LIN {X 0,Y 104.567,Z 489.465,A -85,B 0,C 180,E1 -28252.275,E2 -28252.275} C_VEL
LIN {X 0,Y 104.619,Z 487.581,A -85,B 0,C 180,E1 -28260,E2 -28260} C_VEL
LIN {X 0,Y 104.221,Z 489.218,A -85,B 0,C 180,E1 -28267.958,E2 -28267.958} C_VEL
LIN {X 0,Y 104.511,Z 490.279,A -85,B 0,C 180,E1 -28271.639,E2 -28271.639} C_VEL
LIN {X 0,Y 105.02,Z 492.985,A -85,B 0,C 180,E1 -28277.526,E2 -28277.526} C_VEL
LIN {X 0,Y 105.625,Z 496.885,A -85,B 0,C 180,E1 -28283.53,E2 -28283.53} C_VEL
LIN {X 0,Y 106.054,Z 500.091,A -85,B 0,C 180,E1 -28287.638,E2 -28287.638} C_VEL
LIN {X 0,Y 105.786,Z 504.564,A -85,B 0,C 180,E1 -28292.106,E2 -28292.106} C_VEL
LIN {X 0,Y 104.952,Z 508.015,A -85,B 0,C 180,E1 -28294.982,E2 -28294.982} C_VEL
LIN {X 0,Y 103.687,Z 511.068,A -85,B 0,C 180,E1 -28297.21,E2 -28297.21} C_VEL
LIN {X 0,Y 97.623,Z 518.073,A -85,B 0,C 180,E1 -28300.895,E2 -28300.895} C_VEL
LIN {X 0,Y 90.769,Z 524.928,A -85,B 0,C 180,E1 -28305.826,E2 -28305.826} C_VEL
LIN {X 0,Y 83.786,Z 531.001,A -85,B 0,C 180,E1 -28312.143,E2 -28312.143} C_VEL
LIN {X 0,Y 77.697,Z 535.939,A -85,B 0,C 180,E1 -28320.166,E2 -28320.166} C_VEL
LIN {X 0,Y 73.855,Z 538.844,A -85,B 0,C 180,E1 -28327.627,E2 -28327.627} C_VEL
LIN {X 0,Y 72.25,Z 540.013,A -85,B 0,C 180,E1 -28332.13,E2 -28332.13} C_VEL
LIN {X 0,Y 70.44,Z 541.017,A -85,B 0,C 180,E1 -28336.574,E2 -28336.574} C_VEL
LIN {X 0,Y 68.078,Z 541.734,A -85,B 0,C 180,E1 -28341.053,E2 -28341.053} C_VEL
LIN {X 0,Y 63.796,Z 542.259,A -85,B 0,C 180,E1 -28350.796,E2 -28350.796} C_VEL
LIN {X 0,Y 62.993,Z 542.058,A -85,B 0,C 180,E1 -28356.152,E2 -28356.152} C_VEL
LIN {X 0,Y 63.07,Z 541.9,A -85,B 0,C 180,E1 -28357.958,E2 -28357.958} C_VEL
LIN {X 0,Y 65.242,Z 540.489,A -85,B 0,C 180,E1 -28368.855,E2 -28368.855} C_VEL
LIN {X 0,Y 67.337,Z 539.131,A -85,B 0,C 180,E1 -28374.676,E2 -28374.676} C_VEL
LIN {X 0,Y 71.589,Z 536.26,A -85,B 0,C 180,E1 -28382.681,E2 -28382.681} C_VEL
LIN {X 0,Y 76.937,Z 532.366,A -85,B 0,C 180,E1 -28389.75,E2 -28389.75} C_VEL
LIN {X 0,Y 83.424,Z 527.333,A -85,B 0,C 180,E1 -28395.733,E2 -28395.733} C_VEL
LIN {X 0,Y 90.544,Z 520.995,A -85,B 0,C 180,E1 -28400.915,E2 -28400.915} C_VEL
LIN {X 0,Y 98.183,Z 513.072,A -85,B 0,C 180,E1 -28405.405,E2 -28405.405} C_VEL
LIN {X 0,Y 99.078,Z 511.615,A -85,B 0,C 180,E1 -28406.459,E2 -28406.459} C_VEL
LIN {X 0,Y 100.27,Z 508.389,A -85,B 0,C 180,E1 -28409.327,E2 -28409.327} C_VEL
LIN {X 0,Y 100.77,Z 505.026,A -85,B 0,C 180,E1 -28413.044,E2 -28413.044} C_VEL
LIN {X 0,Y 100.847,Z 503.301,A -85,B 0,C 180,E1 -28415.283,E2 -28415.283} C_VEL
LIN {X 0,Y 100.697,Z 500.442,A -85,B 0,C 180,E1 -28419.575,E2 -28419.575} C_VEL
LIN {X 0,Y 100.449,Z 498.224,A -85,B 0,C 180,E1 -28423.748,E2 -28423.748} C_VEL
LIN {X 0,Y 100.261,Z 496.091,A -85,B 0,C 180,E1 -28428.923,E2 -28428.923} C_VEL
LIN {X 0,Y 100.19,Z 494.427,A -85,B 0,C 180,E1 -28435.977,E2 -28435.977} C_VEL
LIN {X 0,Y 100.55,Z 493.814,A -85,B 0,C 180,E1 -28440,E2 -28440} C_VEL
LIN {X 0,Y 100.504,Z 495.591,A -85,B 0,C 180,E1 -28448.039,E2 -28448.039} C_VEL
LIN {X 0,Y 100.795,Z 497.254,A -85,B 0,C 180,E1 -28452.533,E2 -28452.533} C_VEL
LIN {X 0,Y 100.776,Z 500.825,A -85,B 0,C 180,E1 -28458.29,E2 -28458.29} C_VEL
LIN {X 0,Y 100.458,Z 504.199,A -85,B 0,C 180,E1 -28462.433,E2 -28462.433} C_VEL
LIN {X 0,Y 99.769,Z 508.757,A -85,B 0,C 180,E1 -28467.25,E2 -28467.25} C_VEL
LIN {X 0,Y 99.232,Z 511.294,A -85,B 0,C 180,E1 -28469.72,E2 -28469.72} C_VEL
LIN {X 0,Y 95.471,Z 517.656,A -85,B 0,C 180,E1 -28474.089,E2 -28474.089} C_VEL
LIN {X 0,Y 94.466,Z 519.044,A -85,B 0,C 180,E1 -28475.077,E2 -28475.077} C_VEL
LIN {X 0,Y 86.953,Z 526.468,A -85,B 0,C 180,E1 -28479.839,E2 -28479.839} C_VEL
LIN {X 0,Y 80.119,Z 532.433,A -85,B 0,C 180,E1 -28485.431,E2 -28485.431} C_VEL
LIN {X 0,Y 73.999,Z 537.144,A -85,B 0,C 180,E1 -28491.878,E2 -28491.878} C_VEL
LIN {X 0,Y 68.923,Z 540.745,A -85,B 0,C 180,E1 -28499.346,E2 -28499.346} C_VEL
LIN {X 0,Y 66.354,Z 542.607,A -85,B 0,C 180,E1 -28504.933,E2 -28504.933} C_VEL
LIN {X 0,Y 64.454,Z 544.006,A -85,B 0,C 180,E1 -28510.906,E2 -28510.906} C_VEL
LIN {X 0,Y 63.178,Z 545.009,A -85,B 0,C 180,E1 -28517.144,E2 -28517.144} C_VEL
LIN {X 0,Y 62.555,Z 545.622,A -85,B 0,C 180,E1 -28523.549,E2 -28523.549} C_VEL
LIN {X 0,Y 62.607,Z 545.84,A -85,B 0,C 180,E1 -28529.999,E2 -28529.999} C_VEL
LIN {X 0,Y 62.555,Z 545.604,A -85,B 0,C 180,E1 -28536.45,E2 -28536.45} C_VEL
LIN {X 0,Y 63.178,Z 544.978,A -85,B 0,C 180,E1 -28542.854,E2 -28542.854} C_VEL
LIN {X 0,Y 64.454,Z 543.964,A -85,B 0,C 180,E1 -28549.093,E2 -28549.093} C_VEL
LIN {X 0,Y 66.354,Z 542.546,A -85,B 0,C 180,E1 -28555.066,E2 -28555.066} C_VEL
LIN {X 0,Y 70.496,Z 539.586,A -85,B 0,C 180,E1 -28563.251,E2 -28563.251} C_VEL
LIN {X 0,Y 75.884,Z 535.591,A -85,B 0,C 180,E1 -28570.413,E2 -28570.413} C_VEL
LIN {X 0,Y 83.066,Z 529.781,A -85,B 0,C 180,E1 -28577.18,E2 -28577.18} C_VEL
LIN {X 0,Y 90.653,Z 522.755,A -85,B 0,C 180,E1 -28582.621,E2 -28582.621} C_VEL
LIN {X 0,Y 94.453,Z 518.821,A -85,B 0,C 180,E1 -28584.933,E2 -28584.933} C_VEL
LIN {X 0,Y 98.284,Z 512.767,A -85,B 0,C 180,E1 -28589.101,E2 -28589.101} C_VEL
LIN {X 0,Y 99.145,Z 511.116,A -85,B 0,C 180,E1 -28590.251,E2 -28590.251} C_VEL
LIN {X 0,Y 100.191,Z 505.599,A -85,B 0,C 180,E1 -28595.768,E2 -28595.768} C_VEL
LIN {X 0,Y 100.643,Z 500.62,A -85,B 0,C 180,E1 -28601.685,E2 -28601.685} C_VEL
LIN {X 0,Y 100.676,Z 497.884,A -85,B 0,C 180,E1 -28605.858,E2 -28605.858} C_VEL
LIN {X 0,Y 100.608,Z 496.843,A -85,B 0,C 180,E1 -28607.95,E2 -28607.95} C_VEL
LIN {X 0,Y 100.362,Z 495.354,A -85,B 0,C 180,E1 -28611.949,E2 -28611.949} C_VEL
LIN {X 0,Y 100.504,Z 493.432,A -85,B 0,C 180,E1 -28620,E2 -28620} C_VEL
LIN {X 0,Y 100.123,Z 495.688,A -85,B 0,C 180,E1 -28630.672,E2 -28630.672} C_VEL
LIN {X 0,Y 100.345,Z 497.924,A -85,B 0,C 180,E1 -28636.27,E2 -28636.27} C_VEL
LIN {X 0,Y 100.557,Z 501.264,A -85,B 0,C 180,E1 -28642.057,E2 -28642.057} C_VEL
LIN {X 0,Y 100.754,Z 503.161,A -85,B 0,C 180,E1 -28644.933,E2 -28644.933} C_VEL
LIN {X 0,Y 100.621,Z 505.702,A -85,B 0,C 180,E1 -28648.128,E2 -28648.128} C_VEL
LIN {X 0,Y 100.221,Z 508.006,A -85,B 0,C 180,E1 -28650.572,E2 -28650.572} C_VEL
LIN {X 0,Y 99.079,Z 511.301,A -85,B 0,C 180,E1 -28653.546,E2 -28653.546} C_VEL
LIN {X 0,Y 98.267,Z 512.754,A -85,B 0,C 180,E1 -28654.671,E2 -28654.671} C_VEL
LIN {X 0,Y 90.615,Z 520.73,A -85,B 0,C 180,E1 -28659.142,E2 -28659.142} C_VEL
LIN {X 0,Y 83.479,Z 527.131,A -85,B 0,C 180,E1 -28664.307,E2 -28664.307} C_VEL
LIN {X 0,Y 77.003,Z 532.209,A -85,B 0,C 180,E1 -28670.292,E2 -28670.292} C_VEL
LIN {X 0,Y 71.62,Z 536.145,A -85,B 0,C 180,E1 -28677.337,E2 -28677.337} C_VEL
LIN {X 0,Y 67.347,Z 539.048,A -85,B 0,C 180,E1 -28685.329,E2 -28685.329} C_VEL
LIN {X 0,Y 65.243,Z 540.432,A -85,B 0,C 180,E1 -28691.147,E2 -28691.147} C_VEL
LIN {X 0,Y 62.946,Z 542.016,A -85,B 0,C 180,E1 -28703.59,E2 -28703.59} C_VEL
LIN {X 0,Y 62.722,Z 542.238,A -85,B 0,C 180,E1 -28710.001,E2 -28710.001} C_VEL
LIN {X 0,Y 63.07,Z 541.9,A -85,B 0,C 180,E1 -28717.958,E2 -28717.958} C_VEL
LIN {X 0,Y 63.164,Z 541.44,A -85,B 0,C 180,E1 -28723.3,E2 -28723.3} C_VEL
LIN {X 0,Y 62.614,Z 540.133,A -85,B 0,C 180,E1 -28732.261,E2 -28732.261} C_VEL
LIN {X 0,Y 63.051,Z 538.603,A -85,B 0,C 180,E1 -28739.398,E2 -28739.398} C_VEL
LIN {X 0,Y 64.697,Z 537.117,A -85,B 0,C 180,E1 -28744.344,E2 -28744.344} C_VEL
LIN {X 0,Y 65.581,Z 536.545,A -85,B 0,C 180,E1 -28745.825,E2 -28745.825} C_VEL
LIN {X 0,Y 71.62,Z 532.569,A -85,B 0,C 180,E1 -28753.386,E2 -28753.386} C_VEL
LIN {X 0,Y 78.634,Z 527.536,A -85,B 0,C 180,E1 -28759.438,E2 -28759.438} C_VEL
LIN {X 0,Y 86.239,Z 521.198,A -85,B 0,C 180,E1 -28764.583,E2 -28764.583} C_VEL
LIN {X 0,Y 92.961,Z 514.746,A -85,B 0,C 180,E1 -28768.269,E2 -28768.269} C_VEL
LIN {X 0,Y 93.937,Z 513.296,A -85,B 0,C 180,E1 -28769.361,E2 -28769.361} C_VEL
LIN {X 0,Y 95.048,Z 510.36,A -85,B 0,C 180,E1 -28772.537,E2 -28772.537} C_VEL
LIN {X 0,Y 95.505,Z 507.367,A -85,B 0,C 180,E1 -28776.725,E2 -28776.725} C_VEL
LIN {X 0,Y 95.602,Z 505.021,A -85,B 0,C 180,E1 -28780.682,E2 -28780.682} C_VEL
LIN {X 0,Y 95.508,Z 502.188,A -85,B 0,C 180,E1 -28787.246,E2 -28787.246} C_VEL
LIN {X 0,Y 95.59,Z 500.834,A -85,B 0,C 180,E1 -28791.544,E2 -28791.544} C_VEL
LIN {X 0,Y 96.119,Z 499.403,A -85,B 0,C 180,E1 -28800,E2 -28800} C_VEL
LIN {X 0,Y 95.939,Z 501.238,A -85,B 0,C 180,E1 -28808.425,E2 -28808.425} C_VEL
LIN {X 0,Y 96.016,Z 502.803,A -85,B 0,C 180,E1 -28812.685,E2 -28812.685} C_VEL
LIN {X 0,Y 95.698,Z 505.559,A -85,B 0,C 180,E1 -28817.307,E2 -28817.307} C_VEL
LIN {X 0,Y 94.841,Z 509.862,A -85,B 0,C 180,E1 -28822.931,E2 -28822.931} C_VEL
LIN {X 0,Y 93.951,Z 513.153,A -85,B 0,C 180,E1 -28826.669,E2 -28826.669} C_VEL
LIN {X 0,Y 93.225,Z 514.714,A -85,B 0,C 180,E1 -28828.108,E2 -28828.108} C_VEL
LIN {X 0,Y 89.204,Z 520.202,A -85,B 0,C 180,E1 -28832.117,E2 -28832.117} C_VEL
LIN {X 0,Y 81.283,Z 527.379,A -85,B 0,C 180,E1 -28836.889,E2 -28836.889} C_VEL
LIN {X 0,Y 72.875,Z 533.919,A -85,B 0,C 180,E1 -28843.672,E2 -28843.672} C_VEL
LIN {X 0,Y 66.537,Z 538.248,A -85,B 0,C 180,E1 -28850.671,E2 -28850.671} C_VEL
LIN {X 0,Y 62.904,Z 540.542,A -85,B 0,C 180,E1 -28856.038,E2 -28856.038} C_VEL
LIN {X 0,Y 59.958,Z 542.402,A -85,B 0,C 180,E1 -28862.039,E2 -28862.039} C_VEL
LIN {X 0,Y 57.764,Z 543.802,A -85,B 0,C 180,E1 -28868.591,E2 -28868.591} C_VEL
LIN {X 0,Y 56.267,Z 544.805,A -85,B 0,C 180,E1 -28875.533,E2 -28875.533} C_VEL
LIN {X 0,Y 55.513,Z 545.419,A -85,B 0,C 180,E1 -28882.726,E2 -28882.726} C_VEL
LIN {X 0,Y 55.506,Z 545.636,A -85,B 0,C 180,E1 -28889.999,E2 -28889.999} C_VEL
LIN {X 0,Y 55.513,Z 545.4,A -85,B 0,C 180,E1 -28897.273,E2 -28897.273} C_VEL
LIN {X 0,Y 56.266,Z 544.774,A -85,B 0,C 180,E1 -28904.466,E2 -28904.466} C_VEL
LIN {X 0,Y 57.763,Z 543.759,A -85,B 0,C 180,E1 -28911.407,E2 -28911.407} C_VEL
LIN {X 0,Y 59.957,Z 542.34,A -85,B 0,C 180,E1 -28917.96,E2 -28917.96} C_VEL
LIN {X 0,Y 64.666,Z 539.381,A -85,B 0,C 180,E1 -28926.708,E2 -28926.708} C_VEL
LIN {X 0,Y 70.612,Z 535.385,A -85,B 0,C 180,E1 -28934.163,E2 -28934.163} C_VEL
LIN {X 0,Y 77.727,Z 530.116,A -85,B 0,C 180,E1 -28940.508,E2 -28940.508} C_VEL
LIN {X 0,Y 85.172,Z 523.786,A -85,B 0,C 180,E1 -28945.603,E2 -28945.603} C_VEL
LIN {X 0,Y 89.206,Z 519.977,A -85,B 0,C 180,E1 -28947.878,E2 -28947.878} C_VEL
LIN {X 0,Y 93.154,Z 514.542,A -85,B 0,C 180,E1 -28951.851,E2 -28951.851} C_VEL
LIN {X 0,Y 93.986,Z 512.505,A -85,B 0,C 180,E1 -28953.808,E2 -28953.808} C_VEL
LIN {X 0,Y 94.959,Z 508.635,A -85,B 0,C 180,E1 -28958.281,E2 -28958.281} C_VEL
LIN {X 0,Y 95.621,Z 505.185,A -85,B 0,C 180,E1 -28962.903,E2 -28962.903} C_VEL
LIN {X 0,Y 95.861,Z 502.629,A -85,B 0,C 180,E1 -28967.294,E2 -28967.294} C_VEL
LIN {X 0,Y 95.811,Z 501.022,A -85,B 0,C 180,E1 -28971.564,E2 -28971.564} C_VEL
LIN {X 0,Y 96.077,Z 499.049,A -85,B 0,C 180,E1 -28980,E2 -28980} C_VEL
LIN {X 0,Y 95.454,Z 500.606,A -85,B 0,C 180,E1 -28988.468,E2 -28988.468} C_VEL
LIN {X 0,Y 95.419,Z 501.903,A -85,B 0,C 180,E1 -28992.766,E2 -28992.766} C_VEL
LIN {X 0,Y 95.481,Z 503.704,A -85,B 0,C 180,E1 -28997.123,E2 -28997.123} C_VEL
LIN {X 0,Y 95.413,Z 507.066,A -85,B 0,C 180,E1 -29003.237,E2 -29003.237} C_VEL
LIN {X 0,Y 94.965,Z 510.027,A -85,B 0,C 180,E1 -29007.368,E2 -29007.368} C_VEL
LIN {X 0,Y 93.926,Z 512.988,A -85,B 0,C 180,E1 -29010.634,E2 -29010.634} C_VEL
LIN {X 0,Y 93.045,Z 514.438,A -85,B 0,C 180,E1 -29011.82,E2 -29011.82} C_VEL
LIN {X 0,Y 85.016,Z 522.098,A -85,B 0,C 180,E1 -29016.294,E2 -29016.294} C_VEL
LIN {X 0,Y 78.686,Z 527.336,A -85,B 0,C 180,E1 -29020.607,E2 -29020.607} C_VEL
LIN {X 0,Y 71.678,Z 532.414,A -85,B 0,C 180,E1 -29026.659,E2 -29026.659} C_VEL
LIN {X 0,Y 65.752,Z 536.35,A -85,B 0,C 180,E1 -29033.994,E2 -29033.994} C_VEL
LIN {X 0,Y 60.975,Z 539.253,A -85,B 0,C 180,E1 -29042.546,E2 -29042.546} C_VEL
LIN {X 0,Y 58.573,Z 540.636,A -85,B 0,C 180,E1 -29048.903,E2 -29048.903} C_VEL
LIN {X 0,Y 55.913,Z 542.22,A -85,B 0,C 180,E1 -29062.78,E2 -29062.78} C_VEL
LIN {X 0,Y 55.649,Z 542.442,A -85,B 0,C 180,E1 -29070.001,E2 -29070.001} C_VEL
LIN {X 0,Y 56.027,Z 542.132,A -85,B 0,C 180,E1 -29078.612,E2 -29078.612} C_VEL
LIN {X 0,Y 58.572,Z 540.693,A -85,B 0,C 180,E1 -29091.099,E2 -29091.099} C_VEL
LIN {X 0,Y 60.964,Z 539.335,A -85,B 0,C 180,E1 -29097.461,E2 -29097.461} C_VEL
LIN {X 0,Y 65.581,Z 536.545,A -85,B 0,C 180,E1 -29105.825,E2 -29105.825} C_VEL
LIN {X 0,Y 68.092,Z 534.76,A -85,B 0,C 180,E1 -29110.144,E2 -29110.144} C_VEL
LIN {X 0,Y 71.442,Z 531.374,A -85,B 0,C 180,E1 -29117.28,E2 -29117.28} C_VEL
LIN {X 0,Y 75.447,Z 527.253,A -85,B 0,C 180,E1 -29123.6,E2 -29123.6} C_VEL
LIN {X 0,Y 78.783,Z 524.314,A -85,B 0,C 180,E1 -29126.507,E2 -29126.507} C_VEL
LIN {X 0,Y 86.93,Z 517.296,A -85,B 0,C 180,E1 -29130.982,E2 -29130.982} C_VEL
LIN {X 0,Y 87.982,Z 516.306,A -85,B 0,C 180,E1 -29131.485,E2 -29131.485} C_VEL
LIN {X 0,Y 88.927,Z 515.024,A -85,B 0,C 180,E1 -29132.676,E2 -29132.676} C_VEL
LIN {X 0,Y 89.515,Z 513.597,A -85,B 0,C 180,E1 -29134.476,E2 -29134.476} C_VEL
LIN {X 0,Y 90.136,Z 510.701,A -85,B 0,C 180,E1 -29139.336,E2 -29139.336} C_VEL
LIN {X 0,Y 90.32,Z 509.42,A -85,B 0,C 180,E1 -29141.865,E2 -29141.865} C_VEL
LIN {X 0,Y 90.439,Z 507.624,A -85,B 0,C 180,E1 -29146.518,E2 -29146.518} C_VEL
LIN {X 0,Y 90.643,Z 506.202,A -85,B 0,C 180,E1 -29151.079,E2 -29151.079} C_VEL
LIN {X 0,Y 90.874,Z 505.331,A -85,B 0,C 180,E1 -29155.564,E2 -29155.564} C_VEL
LIN {X 0,Y 91.365,Z 504.752,A -85,B 0,C 180,E1 -29160,E2 -29160} C_VEL
LIN {X 0,Y 91.053,Z 505.547,A -85,B 0,C 180,E1 -29164.427,E2 -29164.427} C_VEL
LIN {X 0,Y 90.996,Z 506.636,A -85,B 0,C 180,E1 -29168.886,E2 -29168.886} C_VEL
LIN {X 0,Y 90.769,Z 508.475,A -85,B 0,C 180,E1 -29173.431,E2 -29173.431} C_VEL
LIN {X 0,Y 90,Z 511.327,A -85,B 0,C 180,E1 -29178.201,E2 -29178.201} C_VEL
LIN {X 0,Y 89.17,Z 514.029,A -85,B 0,C 180,E1 -29181.984,E2 -29181.984} C_VEL
LIN {X 0,Y 88.135,Z 516.54,A -85,B 0,C 180,E1 -29185.046,E2 -29185.046} C_VEL
LIN {X 0,Y 85.447,Z 519.989,A -85,B 0,C 180,E1 -29187.847,E2 -29187.847} C_VEL
LIN {X 0,Y 82.774,Z 522.55,A -85,B 0,C 180,E1 -29189.507,E2 -29189.507} C_VEL
LIN {X 0,Y 74.05,Z 529.57,A -85,B 0,C 180,E1 -29194.712,E2 -29194.712} C_VEL
LIN {X 0,Y 65.694,Z 535.301,A -85,B 0,C 180,E1 -29201.507,E2 -29201.507} C_VEL
LIN {X 0,Y 59.098,Z 539.264,A -85,B 0,C 180,E1 -29209.15,E2 -29209.15} C_VEL
LIN {X 0,Y 53.753,Z 542.197,A -85,B 0,C 180,E1 -29218.466,E2 -29218.466} C_VEL
LIN {X 0,Y 51.176,Z 543.597,A -85,B 0,C 180,E1 -29225.669,E2 -29225.669} C_VEL
LIN {X 0,Y 48.473,Z 545.215,A -85,B 0,C 180,E1 -29241.663,E2 -29241.663} C_VEL
LIN {X 0,Y 48.423,Z 545.433,A -85,B 0,C 180,E1 -29249.999,E2 -29249.999} C_VEL
LIN {X 0,Y 48.473,Z 545.195,A -85,B 0,C 180,E1 -29258.336,E2 -29258.336} C_VEL
LIN {X 0,Y 51.176,Z 543.553,A -85,B 0,C 180,E1 -29274.329,E2 -29274.329} C_VEL
LIN {X 0,Y 53.752,Z 542.134,A -85,B 0,C 180,E1 -29281.533,E2 -29281.533} C_VEL
LIN {X 0,Y 59.097,Z 539.175,A -85,B 0,C 180,E1 -29290.849,E2 -29290.849} C_VEL
LIN {X 0,Y 65.693,Z 535.179,A -85,B 0,C 180,E1 -29298.492,E2 -29298.492} C_VEL
LIN {X 0,Y 74.058,Z 529.393,A -85,B 0,C 180,E1 -29305.293,E2 -29305.293} C_VEL
LIN {X 0,Y 82.772,Z 522.341,A -85,B 0,C 180,E1 -29310.494,E2 -29310.494} C_VEL
LIN {X 0,Y 84.2,Z 521.104,A -85,B 0,C 180,E1 -29311.212,E2 -29311.212} C_VEL
LIN {X 0,Y 87.346,Z 517.408,A -85,B 0,C 180,E1 -29314.04,E2 -29314.04} C_VEL
LIN {X 0,Y 88.064,Z 516.36,A -85,B 0,C 180,E1 -29314.916,E2 -29314.916} C_VEL
LIN {X 0,Y 89.42,Z 512.86,A -85,B 0,C 180,E1 -29319.29,E2 -29319.29} C_VEL
LIN {X 0,Y 90.24,Z 510.135,A -85,B 0,C 180,E1 -29323.247,E2 -29323.247} C_VEL
LIN {X 0,Y 90.654,Z 508.275,A -85,B 0,C 180,E1 -29326.551,E2 -29326.551} C_VEL
LIN {X 0,Y 90.859,Z 506.452,A -85,B 0,C 180,E1 -29331.101,E2 -29331.101} C_VEL
LIN {X 0,Y 91.329,Z 504.437,A -85,B 0,C 180,E1 -29340,E2 -29340} C_VEL
LIN {X 0,Y 90.512,Z 505.989,A -85,B 0,C 180,E1 -29348.934,E2 -29348.934} C_VEL
LIN {X 0,Y 90.364,Z 507.349,A -85,B 0,C 180,E1 -29353.493,E2 -29353.493} C_VEL
LIN {X 0,Y 90.184,Z 509.226,A -85,B 0,C 180,E1 -29358.163,E2 -29358.163} C_VEL
LIN {X 0,Y 89.852,Z 511.77,A -85,B 0,C 180,E1 -29363.022,E2 -29363.022} C_VEL
LIN {X 0,Y 89.399,Z 513.431,A -85,B 0,C 180,E1 -29365.619,E2 -29365.619} C_VEL
LIN {X 0,Y 88.853,Z 514.822,A -85,B 0,C 180,E1 -29367.398,E2 -29367.398} C_VEL
LIN {X 0,Y 88.07,Z 516.02,A -85,B 0,C 180,E1 -29368.622,E2 -29368.622} C_VEL
LIN {X 0,Y 79.665,Z 523.412,A -85,B 0,C 180,E1 -29373.063,E2 -29373.063} C_VEL
LIN {X 0,Y 71.658,Z 529.348,A -85,B 0,C 180,E1 -29378.316,E2 -29378.316} C_VEL
LIN {X 0,Y 64.403,Z 534.034,A -85,B 0,C 180,E1 -29384.822,E2 -29384.822} C_VEL
LIN {X 0,Y 58.198,Z 537.612,A -85,B 0,C 180,E1 -29392.858,E2 -29392.858} C_VEL
LIN {X 0,Y 54.758,Z 539.458,A -85,B 0,C 180,E1 -29399.111,E2 -29399.111} C_VEL
LIN {X 0,Y 50.039,Z 541.823,A -85,B 0,C 180,E1 -29413.687,E2 -29413.687} C_VEL
LIN {X 0,Y 48.877,Z 542.424,A -85,B 0,C 180,E1 -29421.734,E2 -29421.734} C_VEL
LIN {X 0,Y 48.564,Z 542.645,A -85,B 0,C 180,E1 -29430.001,E2 -29430.001} C_VEL
LIN {X 0,Y 48.875,Z 542.449,A -85,B 0,C 180,E1 -29438.268,E2 -29438.268} C_VEL
LIN {X 0,Y 50.039,Z 541.863,A -85,B 0,C 180,E1 -29446.315,E2 -29446.315} C_VEL
LIN {X 0,Y 54.746,Z 539.539,A -85,B 0,C 180,E1 -29460.898,E2 -29460.898} C_VEL
LIN {X 0,Y 60.122,Z 536.667,A -85,B 0,C 180,E1 -29470.012,E2 -29470.012} C_VEL
LIN {X 0,Y 66.641,Z 532.772,A -85,B 0,C 180,E1 -29477.581,E2 -29477.581} C_VEL
LIN {X 0,Y 74.216,Z 527.738,A -85,B 0,C 180,E1 -29483.604,E2 -29483.604} C_VEL
LIN {X 0,Y 78.783,Z 524.314,A -85,B 0,C 180,E1 -29486.507,E2 -29486.507} C_VEL
LIN {X 0,Y 80.877,Z 522.32,A -85,B 0,C 180,E1 -29488.436,E2 -29488.436} C_VEL
LIN {X 0,Y 82.59,Z 519.877,A -85,B 0,C 180,E1 -29491.553,E2 -29491.553} C_VEL
LIN {X 0,Y 83.723,Z 517.203,A -85,B 0,C 180,E1 -29495.915,E2 -29495.915} C_VEL
LIN {X 0,Y 84.374,Z 515.292,A -85,B 0,C 180,E1 -29499.501,E2 -29499.501} C_VEL
LIN {X 0,Y 84.598,Z 514.73,A -85,B 0,C 180,E1 -29500.591,E2 -29500.591} C_VEL
LIN {X 0,Y 84.998,Z 512.773,A -85,B 0,C 180,E1 -29505.637,E2 -29505.637} C_VEL
LIN {X 0,Y 85.402,Z 511.222,A -85,B 0,C 180,E1 -29510.942,E2 -29510.942} C_VEL
LIN {X 0,Y 85.741,Z 510.372,A -85,B 0,C 180,E1 -29515.298,E2 -29515.298} C_VEL
LIN {X 0,Y 86.298,Z 509.788,A -85,B 0,C 180,E1 -29520,E2 -29520} C_VEL
LIN {X 0,Y 85.924,Z 510.6,A -85,B 0,C 180,E1 -29524.691,E2 -29524.691} C_VEL
LIN {X 0,Y 85.62,Z 512.023,A -85,B 0,C 180,E1 -29529.931,E2 -29529.931} C_VEL
LIN {X 0,Y 85.061,Z 513.916,A -85,B 0,C 180,E1 -29534.351,E2 -29534.351} C_VEL
LIN {X 0,Y 83.758,Z 517.069,A -85,B 0,C 180,E1 -29539.611,E2 -29539.611} C_VEL
LIN {X 0,Y 83.068,Z 518.364,A -85,B 0,C 180,E1 -29541.461,E2 -29541.461} C_VEL
LIN {X 0,Y 82.103,Z 519.767,A -85,B 0,C 180,E1 -29543.043,E2 -29543.043} C_VEL
LIN {X 0,Y 80.877,Z 521.101,A -85,B 0,C 180,E1 -29544.156,E2 -29544.156} C_VEL
LIN {X 0,Y 76.529,Z 524.736,A -85,B 0,C 180,E1 -29546.44,E2 -29546.44} C_VEL
LIN {X 0,Y 66.571,Z 531.822,A -85,B 0,C 180,E1 -29552.373,E2 -29552.373} C_VEL
LIN {X 0,Y 58.652,Z 536.532,A -85,B 0,C 180,E1 -29558.842,E2 -29558.842} C_VEL
LIN {X 0,Y 51.721,Z 540.135,A -85,B 0,C 180,E1 -29567.2,E2 -29567.2} C_VEL
LIN {X 0,Y 47.813,Z 541.993,A -85,B 0,C 180,E1 -29573.987,E2 -29573.987} C_VEL
LIN {X 0,Y 42.609,Z 544.395,A -85,B 0,C 180,E1 -29590.737,E2 -29590.737} C_VEL
LIN {X 0,Y 41.447,Z 545.01,A -85,B 0,C 180,E1 -29600.236,E2 -29600.236} C_VEL
LIN {X 0,Y 41.323,Z 545.229,A -85,B 0,C 180,E1 -29609.999,E2 -29609.999} C_VEL
LIN {X 0,Y 41.447,Z 544.991,A -85,B 0,C 180,E1 -29619.762,E2 -29619.762} C_VEL
LIN {X 0,Y 44.768,Z 543.348,A -85,B 0,C 180,E1 -29638.096,E2 -29638.096} C_VEL
LIN {X 0,Y 47.812,Z 541.928,A -85,B 0,C 180,E1 -29646.012,E2 -29646.012} C_VEL
LIN {X 0,Y 53.906,Z 538.969,A -85,B 0,C 180,E1 -29655.811,E2 -29655.811} C_VEL
LIN {X 0,Y 61.211,Z 534.974,A -85,B 0,C 180,E1 -29663.485,E2 -29663.485} C_VEL
LIN {X 0,Y 69.598,Z 529.65,A -85,B 0,C 180,E1 -29669.676,E2 -29669.676} C_VEL
LIN {X 0,Y 78.011,Z 523.372,A -85,B 0,C 180,E1 -29674.276,E2 -29674.276} C_VEL
LIN {X 0,Y 80.842,Z 520.885,A -85,B 0,C 180,E1 -29675.896,E2 -29675.896} C_VEL
LIN {X 0,Y 82.087,Z 519.531,A -85,B 0,C 180,E1 -29676.981,E2 -29676.981} C_VEL
LIN {X 0,Y 83.037,Z 518.126,A -85,B 0,C 180,E1 -29678.592,E2 -29678.592} C_VEL
LIN {X 0,Y 84.417,Z 515.148,A -85,B 0,C 180,E1 -29683.059,E2 -29683.059} C_VEL
LIN {X 0,Y 84.993,Z 513.709,A -85,B 0,C 180,E1 -29685.637,E2 -29685.637} C_VEL
LIN {X 0,Y 85.536,Z 511.672,A -85,B 0,C 180,E1 -29690.542,E2 -29690.542} C_VEL
LIN {X 0,Y 85.833,Z 510.383,A -85,B 0,C 180,E1 -29695.304,E2 -29695.304} C_VEL
LIN {X 0,Y 86.274,Z 509.503,A -85,B 0,C 180,E1 -29700,E2 -29700} C_VEL
LIN {X 0,Y 85.268,Z 511.105,A -85,B 0,C 180,E1 -29709.488,E2 -29709.488} C_VEL
LIN {X 0,Y 84.751,Z 513.424,A -85,B 0,C 180,E1 -29716.873,E2 -29716.873} C_VEL
LIN {X 0,Y 83.928,Z 516.297,A -85,B 0,C 180,E1 -29722.91,E2 -29722.91} C_VEL
LIN {X 0,Y 83.364,Z 517.544,A -85,B 0,C 180,E1 -29724.931,E2 -29724.931} C_VEL
LIN {X 0,Y 74.592,Z 524.727,A -85,B 0,C 180,E1 -29729.365,E2 -29729.365} C_VEL
LIN {X 0,Y 67.487,Z 529.553,A -85,B 0,C 180,E1 -29733.581,E2 -29733.581} C_VEL
LIN {X 0,Y 59.606,Z 534.239,A -85,B 0,C 180,E1 -29739.97,E2 -29739.97} C_VEL
LIN {X 0,Y 52.714,Z 537.817,A -85,B 0,C 180,E1 -29748.194,E2 -29748.194} C_VEL
LIN {X 0,Y 48.795,Z 539.663,A -85,B 0,C 180,E1 -29754.822,E2 -29754.822} C_VEL
LIN {X 0,Y 43.274,Z 542.028,A -85,B 0,C 180,E1 -29771.047,E2 -29771.047} C_VEL
LIN {X 0,Y 41.88,Z 542.628,A -85,B 0,C 180,E1 -29780.34,E2 -29780.34} C_VEL
LIN {X 0,Y 41.469,Z 542.849,A -85,B 0,C 180,E1 -29790.001,E2 -29790.001} C_VEL
LIN {X 0,Y 41.878,Z 542.652,A -85,B 0,C 180,E1 -29799.662,E2 -29799.662} C_VEL
LIN {X 0,Y 43.274,Z 542.067,A -85,B 0,C 180,E1 -29808.955,E2 -29808.955} C_VEL
LIN {X 0,Y 48.783,Z 539.742,A -85,B 0,C 180,E1 -29825.189,E2 -29825.189} C_VEL
LIN {X 0,Y 54.873,Z 536.87,A -85,B 0,C 180,E1 -29834.785,E2 -29834.785} C_VEL
LIN {X 0,Y 62.078,Z 532.975,A -85,B 0,C 180,E1 -29842.42,E2 -29842.42} C_VEL
LIN {X 0,Y 70.239,Z 527.941,A -85,B 0,C 180,E1 -29848.267,E2 -29848.267} C_VEL
LIN {X 0,Y 78.864,Z 521.602,A -85,B 0,C 180,E1 -29853.02,E2 -29853.02} C_VEL
LIN {X 0,Y 83.17,Z 517.985,A -85,B 0,C 180,E1 -29855.007,E2 -29855.007} C_VEL
LIN {X 0,Y 83.981,Z 516.567,A -85,B 0,C 180,E1 -29857.007,E2 -29857.007} C_VEL
LIN {X 0,Y 84.374,Z 515.292,A -85,B 0,C 180,E1 -29859.501,E2 -29859.501} C_VEL
LIN {X 0,Y 84.593,Z 514.229,A -85,B 0,C 180,E1 -29862.081,E2 -29862.081} C_VEL
LIN {X 0,Y 84.196,Z 513.395,A -85,B 0,C 180,E1 -29866.078,E2 -29866.078} C_VEL
LIN {X 0,Y 83.295,Z 513.271,A -85,B 0,C 180,E1 -29870.14,E2 -29870.14} C_VEL
LIN {X 0,Y 81.825,Z 513.852,A -85,B 0,C 180,E1 -29875.798,E2 -29875.798} C_VEL
LIN {X 0,Y 80.73,Z 514.822,A -85,B 0,C 180,E1 -29881.575,E2 -29881.575} C_VEL
LIN {X 0,Y 80.466,Z 515.417,A -85,B 0,C 180,E1 -29885.01,E2 -29885.01} C_VEL
LIN {X 0,Y 79.951,Z 516.823,A -85,B 0,C 180,E1 -29890.126,E2 -29890.126} C_VEL
LIN {X 0,Y 79.419,Z 518.017,A -85,B 0,C 180,E1 -29893.236,E2 -29893.236} C_VEL
LIN {X 0,Y 78.794,Z 519.169,A -85,B 0,C 180,E1 -29895.52,E2 -29895.52} C_VEL
LIN {X 0,Y 77.771,Z 520.866,A -85,B 0,C 180,E1 -29898.424,E2 -29898.424} C_VEL
LIN {X 0,Y 76.67,Z 522.141,A -85,B 0,C 180,E1 -29900.03,E2 -29900.03} C_VEL
LIN {X 0,Y 70.536,Z 526.768,A -85,B 0,C 180,E1 -29902.831,E2 -29902.831} C_VEL
LIN {X 0,Y 60.136,Z 533.309,A -85,B 0,C 180,E1 -29908.773,E2 -29908.773} C_VEL
LIN {X 0,Y 51.788,Z 537.635,A -85,B 0,C 180,E1 -29915.486,E2 -29915.486} C_VEL
LIN {X 0,Y 46.753,Z 539.931,A -85,B 0,C 180,E1 -29921.269,E2 -29921.269} C_VEL
LIN {X 0,Y 42.249,Z 541.788,A -85,B 0,C 180,E1 -29928.287,E2 -29928.287} C_VEL
LIN {X 0,Y 35.969,Z 544.191,A -85,B 0,C 180,E1 -29946.995,E2 -29946.995} C_VEL
LIN {X 0,Y 34.469,Z 544.807,A -85,B 0,C 180,E1 -29958.234,E2 -29958.234} C_VEL
LIN {X 0,Y 34.237,Z 545.025,A -85,B 0,C 180,E1 -29969.999,E2 -29969.999} C_VEL
LIN {X 0,Y 34.469,Z 544.786,A -85,B 0,C 180,E1 -29981.764,E2 -29981.764} C_VEL
LIN {X 0,Y 38.625,Z 543.142,A -85,B 0,C 180,E1 -30003.082,E2 -30003.082} C_VEL
LIN {X 0,Y 42.248,Z 541.722,A -85,B 0,C 180,E1 -30011.712,E2 -30011.712} C_VEL
LIN {X 0,Y 49.205,Z 538.764,A -85,B 0,C 180,E1 -30021.772,E2 -30021.772} C_VEL
LIN {X 0,Y 57.266,Z 534.768,A -85,B 0,C 180,E1 -30029.212,E2 -30029.212} C_VEL
LIN {X 0,Y 66.372,Z 529.387,A -85,B 0,C 180,E1 -30035.047,E2 -30035.047} C_VEL
LIN {X 0,Y 75.187,Z 523.165,A -85,B 0,C 180,E1 -30039.184,E2 -30039.184} C_VEL
LIN {X 0,Y 77.177,Z 521.384,A -85,B 0,C 180,E1 -30040.563,E2 -30040.563} C_VEL
LIN {X 0,Y 77.975,Z 520.311,A -85,B 0,C 180,E1 -30042.15,E2 -30042.15} C_VEL
LIN {X 0,Y 79.395,Z 517.771,A -85,B 0,C 180,E1 -30046.832,E2 -30046.832} C_VEL
LIN {X 0,Y 79.833,Z 516.663,A -85,B 0,C 180,E1 -30049.859,E2 -30049.859} C_VEL
LIN {X 0,Y 80.371,Z 515.221,A -85,B 0,C 180,E1 -30054.984,E2 -30054.984} C_VEL
LIN {X 0,Y 80.924,Z 514.29,A -85,B 0,C 180,E1 -30060,E2 -30060} C_VEL
LIN {X 0,Y 79.843,Z 515.488,A -85,B 0,C 180,E1 -30067.679,E2 -30067.679} C_VEL
LIN {X 0,Y 79.395,Z 516.72,A -85,B 0,C 180,E1 -30073.169,E2 -30073.169} C_VEL
LIN {X 0,Y 78.778,Z 518.433,A -85,B 0,C 180,E1 -30078.195,E2 -30078.195} C_VEL
LIN {X 0,Y 78.195,Z 519.691,A -85,B 0,C 180,E1 -30081.071,E2 -30081.071} C_VEL
LIN {X 0,Y 74.396,Z 522.717,A -85,B 0,C 180,E1 -30082.92,E2 -30082.92} C_VEL
LIN {X 0,Y 66.818,Z 527.953,A -85,B 0,C 180,E1 -30086.615,E2 -30086.615} C_VEL
LIN {X 0,Y 58.062,Z 533.03,A -85,B 0,C 180,E1 -30092.081,E2 -30092.081} C_VEL
LIN {X 0,Y 50.114,Z 536.964,A -85,B 0,C 180,E1 -30099.528,E2 -30099.528} C_VEL
LIN {X 0,Y 43.186,Z 539.868,A -85,B 0,C 180,E1 -30109.388,E2 -30109.388} C_VEL
LIN {X 0,Y 39.451,Z 541.25,A -85,B 0,C 180,E1 -30117.695,E2 -30117.695} C_VEL
LIN {X 0,Y 34.897,Z 542.832,A -85,B 0,C 180,E1 -30138.383,E2 -30138.383} C_VEL
LIN {X 0,Y 34.391,Z 543.052,A -85,B 0,C 180,E1 -30150.001,E2 -30150.001} C_VEL
LIN {X 0,Y 34.895,Z 542.856,A -85,B 0,C 180,E1 -30161.62,E2 -30161.62} C_VEL
LIN {X 0,Y 39.448,Z 541.304,A -85,B 0,C 180,E1 -30182.309,E2 -30182.309} C_VEL
LIN {X 0,Y 43.176,Z 539.946,A -85,B 0,C 180,E1 -30190.627,E2 -30190.627} C_VEL
LIN {X 0,Y 50.066,Z 537.074,A -85,B 0,C 180,E1 -30200.54,E2 -30200.54} C_VEL
LIN {X 0,Y 58.027,Z 533.177,A -85,B 0,C 180,E1 -30207.976,E2 -30207.976} C_VEL
LIN {X 0,Y 66.782,Z 528.143,A -85,B 0,C 180,E1 -30213.449,E2 -30213.449} C_VEL
LIN {X 0,Y 75.91,Z 521.804,A -85,B 0,C 180,E1 -30217.796,E2 -30217.796} C_VEL
LIN {X 0,Y 78.261,Z 519.889,A -85,B 0,C 180,E1 -30218.948,E2 -30218.948} C_VEL
LIN {X 0,Y 78.912,Z 518.594,A -85,B 0,C 180,E1 -30221.837,E2 -30221.837} C_VEL
LIN {X 0,Y 79.46,Z 516.978,A -85,B 0,C 180,E1 -30226.638,E2 -30226.638} C_VEL
LIN {X 0,Y 79.765,Z 516.17,A -85,B 0,C 180,E1 -30229.85,E2 -30229.85} C_VEL
LIN {X 0,Y 80.296,Z 515.161,A -85,B 0,C 180,E1 -30234.978,E2 -30234.978} C_VEL
LIN {X 0,Y 80.95,Z 514.548,A -85,B 0,C 180,E1 -30240,E2 -30240} C_VEL
LIN {X 0,Y 80.73,Z 514.822,A -85,B 0,C 180,E1 -30241.575,E2 -30241.575} C_VEL
LIN {X 0,Y 80.046,Z 515.685,A -85,B 0,C 180,E1 -30244.324,E2 -30244.324} C_VEL
LIN {X 0,Y 78.323,Z 517.579,A -85,B 0,C 180,E1 -30247.745,E2 -30247.745} C_VEL
LIN {X 0,Y 75.297,Z 520.67,A -85,B 0,C 180,E1 -30251.756,E2 -30251.756} C_VEL
LIN {X 0,Y 72.473,Z 523.302,A -85,B 0,C 180,E1 -30254.868,E2 -30254.868} C_VEL
LIN {X 0,Y 71.328,Z 524.329,A -85,B 0,C 180,E1 -30256.118,E2 -30256.118} C_VEL
LIN {X 0,Y 60.142,Z 531.414,A -85,B 0,C 180,E1 -30260.792,E2 -30260.792} C_VEL
LIN {X 0,Y 50.936,Z 536.124,A -85,B 0,C 180,E1 -30266.251,E2 -30266.251} C_VEL
LIN {X 0,Y 42.385,Z 539.727,A -85,B 0,C 180,E1 -30273.996,E2 -30273.996} C_VEL
LIN {X 0,Y 37.228,Z 541.584,A -85,B 0,C 180,E1 -30280.961,E2 -30280.961} C_VEL
LIN {X 0,Y 32.889,Z 542.984,A -85,B 0,C 180,E1 -30290.127,E2 -30290.127} C_VEL
LIN {X 0,Y 27.538,Z 544.602,A -85,B 0,C 180,E1 -30315.213,E2 -30315.213} C_VEL
LIN {X 0,Y 27.123,Z 544.82,A -85,B 0,C 180,E1 -30329.998,E2 -30329.998} C_VEL
LIN {X 0,Y 27.538,Z 544.582,A -85,B 0,C 180,E1 -30344.785,E2 -30344.785} C_VEL
LIN {X 0,Y 32.888,Z 542.937,A -85,B 0,C 180,E1 -30369.871,E2 -30369.871} C_VEL
LIN {X 0,Y 37.226,Z 541.517,A -85,B 0,C 180,E1 -30379.038,E2 -30379.038} C_VEL
LIN {X 0,Y 45.144,Z 538.558,A -85,B 0,C 180,E1 -30388.895,E2 -30388.895} C_VEL
LIN {X 0,Y 53.972,Z 534.563,A -85,B 0,C 180,E1 -30395.712,E2 -30395.712} C_VEL
LIN {X 0,Y 63.342,Z 529.399,A -85,B 0,C 180,E1 -30400.707,E2 -30400.707} C_VEL
LIN {X 0,Y 71.324,Z 524.13,A -85,B 0,C 180,E1 -30403.889,E2 -30403.889} C_VEL
LIN {X 0,Y 72.638,Z 522.922,A -85,B 0,C 180,E1 -30405.359,E2 -30405.359} C_VEL
LIN {X 0,Y 73.79,Z 521.285,A -85,B 0,C 180,E1 -30409.019,E2 -30409.019} C_VEL
LIN {X 0,Y 74.609,Z 519.78,A -85,B 0,C 180,E1 -30414.595,E2 -30414.595} C_VEL
LIN {X 0,Y 75.305,Z 518.788,A -85,B 0,C 180,E1 -30420,E2 -30420} C_VEL
LIN {X 0,Y 74.172,Z 519.801,A -85,B 0,C 180,E1 -30427.241,E2 -30427.241} C_VEL
LIN {X 0,Y 73.81,Z 520.455,A -85,B 0,C 180,E1 -30430.979,E2 -30430.979} C_VEL
LIN {X 0,Y 72.969,Z 522.074,A -85,B 0,C 180,E1 -30436.795,E2 -30436.795} C_VEL
LIN {X 0,Y 68.747,Z 525.139,A -85,B 0,C 180,E1 -30438.983,E2 -30438.983} C_VEL
LIN {X 0,Y 60.8,Z 529.964,A -85,B 0,C 180,E1 -30442.372,E2 -30442.372} C_VEL
LIN {X 0,Y 51.646,Z 534.649,A -85,B 0,C 180,E1 -30447.809,E2 -30447.809} C_VEL
LIN {X 0,Y 43.191,Z 538.227,A -85,B 0,C 180,E1 -30455.553,E2 -30455.553} C_VEL
LIN {X 0,Y 38.084,Z 540.072,A -85,B 0,C 180,E1 -30462.426,E2 -30462.426} C_VEL
LIN {X 0,Y 30.2,Z 542.436,A -85,B 0,C 180,E1 -30482.263,E2 -30482.263} C_VEL
LIN {X 0,Y 27.974,Z 543.037,A -85,B 0,C 180,E1 -30495.451,E2 -30495.451} C_VEL
LIN {X 0,Y 27.295,Z 543.256,A -85,B 0,C 180,E1 -30510.002,E2 -30510.002} C_VEL
LIN {X 0,Y 27.973,Z 543.06,A -85,B 0,C 180,E1 -30524.553,E2 -30524.553} C_VEL
LIN {X 0,Y 30.2,Z 542.474,A -85,B 0,C 180,E1 -30537.74,E2 -30537.74} C_VEL
LIN {X 0,Y 38.074,Z 540.149,A -85,B 0,C 180,E1 -30557.592,E2 -30557.592} C_VEL
LIN {X 0,Y 45.873,Z 537.278,A -85,B 0,C 180,E1 -30567.421,E2 -30567.421} C_VEL
LIN {X 0,Y 54.601,Z 533.38,A -85,B 0,C 180,E1 -30574.292,E2 -30574.292} C_VEL
LIN {X 0,Y 63.927,Z 528.345,A -85,B 0,C 180,E1 -30579.145,E2 -30579.145} C_VEL
LIN {X 0,Y 71.847,Z 523.178,A -85,B 0,C 180,E1 -30582.373,E2 -30582.373} C_VEL
LIN {X 0,Y 73.085,Z 522.229,A -85,B 0,C 180,E1 -30583.232,E2 -30583.232} C_VEL
LIN {X 0,Y 73.881,Z 520.644,A -85,B 0,C 180,E1 -30589.032,E2 -30589.032} C_VEL
LIN {X 0,Y 74.562,Z 519.652,A -85,B 0,C 180,E1 -30594.591,E2 -30594.591} C_VEL
LIN {X 0,Y 75.325,Z 519.028,A -85,B 0,C 180,E1 -30600,E2 -30600} C_VEL
LIN {X 0,Y 74.676,Z 519.97,A -85,B 0,C 180,E1 -30605.4,E2 -30605.4} C_VEL
LIN {X 0,Y 73.837,Z 521.475,A -85,B 0,C 180,E1 -30610.974,E2 -30610.974} C_VEL
LIN {X 0,Y 72.473,Z 523.302,A -85,B 0,C 180,E1 -30614.868,E2 -30614.868} C_VEL
LIN {X 0,Y 70.005,Z 525.251,A -85,B 0,C 180,E1 -30616.614,E2 -30616.614} C_VEL
LIN {X 0,Y 66.959,Z 527.27,A -85,B 0,C 180,E1 -30617.675,E2 -30617.675} C_VEL
LIN {X 0,Y 61.773,Z 530.125,A -85,B 0,C 180,E1 -30618.346,E2 -30618.346} C_VEL
LIN {X 0,Y 50.317,Z 535.163,A -85,B 0,C 180,E1 -30618.694,E2 -30618.694} C_VEL
LIN {X 0,Y 46.531,Z 536.649,A -85,B 0,C 180,E1 -30619.73,E2 -30619.73} C_VEL
LIN {X 0,Y 44.735,Z 537.339,A -85,B 0,C 180,E1 -30620.7,E2 -30620.7} C_VEL
LIN {X 0,Y 38.851,Z 539.523,A -85,B 0,C 180,E1 -30625.243,E2 -30625.243} C_VEL
LIN {X 0,Y 32.993,Z 541.379,A -85,B 0,C 180,E1 -30631.562,E2 -30631.562} C_VEL
LIN {X 0,Y 27.792,Z 542.779,A -85,B 0,C 180,E1 -30640.653,E2 -30640.653} C_VEL
LIN {X 0,Y 20.746,Z 544.398,A -85,B 0,C 180,E1 -30670.196,E2 -30670.196} C_VEL
LIN {X 0,Y 20.016,Z 544.616,A -85,B 0,C 180,E1 -30689.998,E2 -30689.998} C_VEL
LIN {X 0,Y 20.745,Z 544.377,A -85,B 0,C 180,E1 -30709.8,E2 -30709.8} C_VEL
LIN {X 0,Y 27.791,Z 542.732,A -85,B 0,C 180,E1 -30739.345,E2 -30739.345} C_VEL
LIN {X 0,Y 32.992,Z 541.311,A -85,B 0,C 180,E1 -30748.437,E2 -30748.437} C_VEL
LIN {X 0,Y 41.909,Z 538.352,A -85,B 0,C 180,E1 -30757.267,E2 -30757.267} C_VEL
LIN {X 0,Y 51.456,Z 534.357,A -85,B 0,C 180,E1 -30762.955,E2 -30762.955} C_VEL
LIN {X 0,Y 62.974,Z 528.215,A -85,B 0,C 180,E1 -30767.55,E2 -30767.55} C_VEL
LIN {X 0,Y 67.152,Z 525.61,A -85,B 0,C 180,E1 -30768.836,E2 -30768.836} C_VEL
LIN {X 0,Y 68.021,Z 524.657,A -85,B 0,C 180,E1 -30771.394,E2 -30771.394} C_VEL
LIN {X 0,Y 68.484,Z 524.014,A -85,B 0,C 180,E1 -30774.11,E2 -30774.11} C_VEL
LIN {X 0,Y 69.41,Z 522.988,A -85,B 0,C 180,E1 -30780,E2 -30780} C_VEL
LIN {X 0,Y 68.325,Z 523.736,A -85,B 0,C 180,E1 -30786.473,E2 -30786.473} C_VEL
LIN {X 0,Y 67.531,Z 524.718,A -85,B 0,C 180,E1 -30792.014,E2 -30792.014} C_VEL
LIN {X 0,Y 65.097,Z 526.368,A -85,B 0,C 180,E1 -30793.675,E2 -30793.675} C_VEL
LIN {X 0,Y 55.192,Z 531.856,A -85,B 0,C 180,E1 -30797.252,E2 -30797.252} C_VEL
LIN {X 0,Y 45.569,Z 536.16,A -85,B 0,C 180,E1 -30802.28,E2 -30802.28} C_VEL
LIN {X 0,Y 39.483,Z 538.432,A -85,B 0,C 180,E1 -30807.127,E2 -30807.127} C_VEL
LIN {X 0,Y 33.702,Z 540.277,A -85,B 0,C 180,E1 -30813.477,E2 -30813.477} C_VEL
LIN {X 0,Y 24.156,Z 542.64,A -85,B 0,C 180,E1 -30834.419,E2 -30834.419} C_VEL
LIN {X 0,Y 20.214,Z 543.46,A -85,B 0,C 180,E1 -30870.002,E2 -30870.002} C_VEL
LIN {X 0,Y 21.184,Z 543.264,A -85,B 0,C 180,E1 -30889.377,E2 -30889.377} C_VEL
LIN {X 0,Y 24.156,Z 542.678,A -85,B 0,C 180,E1 -30905.585,E2 -30905.585} C_VEL
LIN {X 0,Y 33.694,Z 540.352,A -85,B 0,C 180,E1 -30926.55,E2 -30926.55} C_VEL
LIN {X 0,Y 42.468,Z 537.482,A -85,B 0,C 180,E1 -30935.534,E2 -30935.534} C_VEL
LIN {X 0,Y 51.922,Z 533.582,A -85,B 0,C 180,E1 -30941.354,E2 -30941.354} C_VEL
LIN {X 0,Y 61.759,Z 528.548,A -85,B 0,C 180,E1 -30945.305,E2 -30945.305} C_VEL
LIN {X 0,Y 65.072,Z 526.567,A -85,B 0,C 180,E1 -30946.419,E2 -30946.419} C_VEL
LIN {X 0,Y 67.601,Z 524.889,A -85,B 0,C 180,E1 -30947.999,E2 -30947.999} C_VEL
LIN {X 0,Y 68.523,Z 523.795,A -85,B 0,C 180,E1 -30954.113,E2 -30954.113} C_VEL
LIN {X 0,Y 69.423,Z 523.194,A -85,B 0,C 180,E1 -30960,E2 -30960} C_VEL
LIN {X 0,Y 68.523,Z 524.196,A -85,B 0,C 180,E1 -30965.887,E2 -30965.887} C_VEL
LIN {X 0,Y 68.085,Z 524.819,A -85,B 0,C 180,E1 -30968.591,E2 -30968.591} C_VEL
LIN {X 0,Y 67.207,Z 525.778,A -85,B 0,C 180,E1 -30971.153,E2 -30971.153} C_VEL
LIN {X 0,Y 57.989,Z 531.209,A -85,B 0,C 180,E1 -30974.168,E2 -30974.168} C_VEL
LIN {X 0,Y 48.212,Z 535.921,A -85,B 0,C 180,E1 -30978.642,E2 -30978.642} C_VEL
LIN {X 0,Y 44.735,Z 537.339,A -85,B 0,C 180,E1 -30980.7,E2 -30980.7} C_VEL
LIN {X 0,Y 39.522,Z 539.191,A -85,B 0,C 180,E1 -30983.574,E2 -30983.574} C_VEL
LIN {X 0,Y 30.204,Z 541.563,A -85,B 0,C 180,E1 -30987.56,E2 -30987.56} C_VEL
LIN {X 0,Y 22.751,Z 542.93,A -85,B 0,C 180,E1 -30992.866,E2 -30992.866} C_VEL
LIN {X 0,Y 17.799,Z 543.674,A -85,B 0,C 180,E1 -31001.896,E2 -31001.896} C_VEL
LIN {X 0,Y 16.468,Z 543.82,A -85,B 0,C 180,E1 -31006.734,E2 -31006.734} C_VEL
LIN {X 0,Y 12.923,Z 544.412,A -85,B 0,C 180,E1 -31049.997,E2 -31049.997} C_VEL
LIN {X 0,Y 14.25,Z 544.172,A -85,B 0,C 180,E1 -31079.548,E2 -31079.548} C_VEL
LIN {X 0,Y 23.76,Z 542.526,A -85,B 0,C 180,E1 -31112.54,E2 -31112.54} C_VEL
LIN {X 0,Y 29.884,Z 541.105,A -85,B 0,C 180,E1 -31120.164,E2 -31120.164} C_VEL
LIN {X 0,Y 39.703,Z 538.147,A -85,B 0,C 180,E1 -31126.793,E2 -31126.793} C_VEL
LIN {X 0,Y 49.832,Z 534.151,A -85,B 0,C 180,E1 -31130.829,E2 -31130.829} C_VEL
LIN {X 0,Y 60.104,Z 529.014,A -85,B 0,C 180,E1 -31133.635,E2 -31133.635} C_VEL
LIN {X 0,Y 62.488,Z 527.518,A -85,B 0,C 180,E1 -31135.329,E2 -31135.329} C_VEL
LIN {X 0,Y 63.231,Z 526.825,A -85,B 0,C 180,E1 -31140,E2 -31140} C_VEL
LIN {X 0,Y 62.094,Z 527.502,A -85,B 0,C 180,E1 -31146.499,E2 -31146.499} C_VEL
LIN {X 0,Y 59.603,Z 528.973,A -85,B 0,C 180,E1 -31148.428,E2 -31148.428} C_VEL
LIN {X 0,Y 50.119,Z 533.644,A -85,B 0,C 180,E1 -31151.018,E2 -31151.018} C_VEL
LIN {X 0,Y 40.067,Z 537.58,A -85,B 0,C 180,E1 -31155.263,E2 -31155.263} C_VEL
LIN {X 0,Y 30.363,Z 540.482,A -85,B 0,C 180,E1 -31162.205,E2 -31162.205} C_VEL
LIN {X 0,Y 18.838,Z 542.845,A -85,B 0,C 180,E1 -31181.743,E2 -31181.743} C_VEL
LIN {X 0,Y 14.695,Z 543.444,A -85,B 0,C 180,E1 -31201.432,E2 -31201.432} C_VEL
LIN {X 0,Y 13.126,Z 543.664,A -85,B 0,C 180,E1 -31230.003,E2 -31230.003} C_VEL
LIN {X 0,Y 14.695,Z 543.467,A -85,B 0,C 180,E1 -31258.575,E2 -31258.575} C_VEL
LIN {X 0,Y 18.838,Z 542.881,A -85,B 0,C 180,E1 -31278.262,E2 -31278.262} C_VEL
LIN {X 0,Y 30.357,Z 540.556,A -85,B 0,C 180,E1 -31297.832,E2 -31297.832} C_VEL
LIN {X 0,Y 40.051,Z 537.685,A -85,B 0,C 180,E1 -31304.828,E2 -31304.828} C_VEL
LIN {X 0,Y 50.105,Z 533.785,A -85,B 0,C 180,E1 -31309.073,E2 -31309.073} C_VEL
LIN {X 0,Y 59.628,Z 529.129,A -85,B 0,C 180,E1 -31311.674,E2 -31311.674} C_VEL
LIN {X 0,Y 62.173,Z 527.65,A -85,B 0,C 180,E1 -31313.509,E2 -31313.509} C_VEL
LIN {X 0,Y 63.233,Z 527.013,A -85,B 0,C 180,E1 -31320,E2 -31320} C_VEL
LIN {X 0,Y 62.505,Z 527.694,A -85,B 0,C 180,E1 -31324.652,E2 -31324.652} C_VEL
LIN {X 0,Y 60.102,Z 529.186,A -85,B 0,C 180,E1 -31326.328,E2 -31326.328} C_VEL
LIN {X 0,Y 49.834,Z 534.284,A -85,B 0,C 180,E1 -31329.171,E2 -31329.171} C_VEL
LIN {X 0,Y 39.705,Z 538.245,A -85,B 0,C 180,E1 -31333.206,E2 -31333.206} C_VEL
LIN {X 0,Y 29.886,Z 541.175,A -85,B 0,C 180,E1 -31339.835,E2 -31339.835} C_VEL
LIN {X 0,Y 18.307,Z 543.578,A -85,B 0,C 180,E1 -31359.841,E2 -31359.841} C_VEL
LIN {X 0,Y 16.468,Z 543.82,A -85,B 0,C 180,E1 -31366.734,E2 -31366.734} C_VEL
LIN {X 0,Y 14.052,Z 544.158,A -85,B 0,C 180,E1 -31378.381,E2 -31378.381} C_VEL
LIN {X 0,Y 11.824,Z 544.297,A -85,B 0,C 180,E1 -31392.854,E2 -31392.854} C_VEL
LIN {X 0,Y 9.706,Z 544.205,A -85,B 0,C 180,E1 -31434.826,E2 -31434.826} C_VEL
LIN {X 0,Y 13.027,Z 543.652,A -85,B 0,C 180,E1 -31473.092,E2 -31473.092} C_VEL
LIN {X 0,Y 17.923,Z 542.922,A -85,B 0,C 180,E1 -31486.118,E2 -31486.118} C_VEL
LIN {X 0,Y 19.782,Z 542.568,A -85,B 0,C 180,E1 -31488.328,E2 -31488.328} C_VEL
LIN {X 0,Y 28.273,Z 540.9,A -85,B 0,C 180,E1 -31493.873,E2 -31493.873} C_VEL
LIN {X 0,Y 38.702,Z 537.941,A -85,B 0,C 180,E1 -31497.139,E2 -31497.139} C_VEL
LIN {X 0,Y 51.451,Z 532.923,A -85,B 0,C 180,E1 -31499.432,E2 -31499.432} C_VEL
LIN {X 0,Y 56.223,Z 530.631,A -85,B 0,C 180,E1 -31500.087,E2 -31500.087} C_VEL
LIN {X 0,Y 56.254,Z 530.58,A -85,B 0,C 180,E1 -31501.896,E2 -31501.896} C_VEL
LIN {X 0,Y 45.765,Z 535.266,A -85,B 0,C 180,E1 -31503.458,E2 -31503.458} C_VEL
LIN {X 0,Y 35.342,Z 538.842,A -85,B 0,C 180,E1 -31506.131,E2 -31506.131} C_VEL
LIN {X 0,Y 28.448,Z 540.687,A -85,B 0,C 180,E1 -31508.818,E2 -31508.818} C_VEL
LIN {X 0,Y 15.075,Z 543.049,A -85,B 0,C 180,E1 -31521.19,E2 -31521.19} C_VEL
LIN {X 0,Y 9.12,Z 543.648,A -85,B 0,C 180,E1 -31539.596,E2 -31539.596} C_VEL
LIN {X 0,Y 6.027,Z 543.868,A -85,B 0,C 180,E1 -31590.007,E2 -31590.007} C_VEL
LIN {X 0,Y 9.12,Z 543.671,A -85,B 0,C 180,E1 -31640.415,E2 -31640.415} C_VEL
LIN {X 0,Y 15.076,Z 543.085,A -85,B 0,C 180,E1 -31658.816,E2 -31658.816} C_VEL
LIN {X 0,Y 28.445,Z 540.76,A -85,B 0,C 180,E1 -31671.23,E2 -31671.23} C_VEL
LIN {X 0,Y 38.8,Z 537.889,A -85,B 0,C 180,E1 -31675.042,E2 -31675.042} C_VEL
LIN {X 0,Y 51.502,Z 532.996,A -85,B 0,C 180,E1 -31677.575,E2 -31677.575} C_VEL
LIN {X 0,Y 56.253,Z 530.753,A -85,B 0,C 180,E1 -31678.182,E2 -31678.182} C_VEL
LIN {X 0,Y 56.225,Z 530.803,A -85,B 0,C 180,E1 -31679.941,E2 -31679.941} C_VEL
LIN {X 0,Y 45.698,Z 535.514,A -85,B 0,C 180,E1 -31681.482,E2 -31681.482} C_VEL
LIN {X 0,Y 35.218,Z 539.115,A -85,B 0,C 180,E1 -31683.784,E2 -31683.784} C_VEL
LIN {X 0,Y 28.274,Z 540.971,A -85,B 0,C 180,E1 -31686.127,E2 -31686.127} C_VEL
LIN {X 0,Y 14.79,Z 543.373,A -85,B 0,C 180,E1 -31698.122,E2 -31698.122} C_VEL
LIN {X 0,Y 8.795,Z 543.989,A -85,B 0,C 180,E1 -31716.947,E2 -31716.947} C_VEL
LIN {X 0,Y 5.817,Z 544.208,A -85,B 0,C 180,E1 -31769.993,E2 -31769.993} C_VEL
LIN {X 0,Y 8.794,Z 543.968,A -85,B 0,C 180,E1 -31823.048,E2 -31823.048} C_VEL
LIN {X 0,Y 19.782,Z 542.568,A -85,B 0,C 180,E1 -31848.328,E2 -31848.328} C_VEL
LIN {X 0,Y 21.965,Z 544.547,A -85,B 0,C 180,E1 -31850.179,E2 -31850.179} C_VEL
LIN {X 0,Y 21.965,Z 600,A -85,B 0,C 180,E1 -31850.179,E2 -31850.179} C_VEL
LIN {X 0,Y 21.965,Z 600,A -85,B 0,C 180,E1 -31850.179,E2 -31850.179}

QRS_NEXT_CUT()

QRS_NEXT()
QRS_HOME()

END
